// TIA Portal V17 export
// export: Created 2026-04-13T11:12:44.8952859Z, ExportSetting WithDefaults, DisplayName Totally Integrated Automation Portal, DisplayVersion V17 Update 4, DisplayName TIA Portal Openness, DisplayVersion V17 Update 4, DisplayName TIA Portal Version Control Interface, DisplayVersion V17, DisplayName SINAMICS Startdrive Advanced, DisplayVersion V17, DisplayName SINAMICS Startdrive G130, G150, S120, S150, SINAMICS MV, S210, DisplayVersion V17, DisplayName SINAMICS Startdrive G110M, G120, G120C, G120D, G120P, G115D, DisplayVersion V17, DisplayName STEP 7 Professional, DisplayVersion V17 Update 4, DisplayName STEP 7 Safety, DisplayVersion V17, DisplayName WinCC Professional, DisplayVersion V17 Update 4
FUNCTION_BLOCK "Send_Config"   // FB611, SCL
TITLE = Send Configuration
AUTHOR : SIMATIC
FAMILY : Freeport
NAME : SendConf
VERSION : 4.0
// stored: IsIECCheckEnabled false, SetENOAutomatically false, UDAEnableTagReadback false
   VAR_INPUT
      REQ : Bool;   // Startet die Konfiguration für Senden bei steigender Flanke / Activates the configuration for sending on rising edge
      PORT : PORT := 0;   // Kommunikationsport, Hardwarekennung / Communication port, Hardware Identifier
      RTSONDLY : UInt := 16#00;   // Wartezeit nach Aktivierung von RTS, vor Übertragung von Tx-Daten (ms) / Time to wait after activating RTS before transmission will be initiated (ms)
      RTSOFFDLY : UInt := 16#00;   // Wartezeit nach Übertragung von Tx-Daten, bevor RTS deaktiviert wird (ms) / Time to wait before de-activating RTS once transmission has been completed (ms)
      BREAK : UInt := 16#00;   // Pause vor Start jeder Übertragung (Bitzeiten) / On start of a message, a break will be sent for the specified no. of bit times
      IDLELINE : UInt := 16#00;   // Leerlaufzeit vor Start jeder Übertragung (Bitzeiten) / Number of bits times the line will be idle before the next transmission
      USR_END : String[2] := '';   // Anzahl der Endekennzeichen / Number of characters in the end delimiter
      APP_END : String[5] := '';   // Anzahl angehängter Zeichen / Number of characters to be appended to the transmitted message
   END_VAR
   VAR_OUTPUT
      DONE : Bool;   // Anweisung beendet ohne Fehler / Instruction finished without error
      ERROR : Bool;   // Anweisung beendet mit Fehler / Instruction finished with error
      STATUS : Word := W#16#7000;   // Zusätzliche Fehlerinformation / Detailed error information
   END_VAR
   VAR
      b_e_REQ : Bool;   // Flankenbit für REQ / Edge flag for REQ
      y_state : SInt := 16#00;   // Status der Anweisung / State of instruction
      WRREC { S7_SetPoint := 'True'} : WRREC;   // Lokale Instanz der Anweisung WRREC / Local instance of instruction WRREC
      RDREC { S7_SetPoint := 'True'} : RDREC;   // Lokale Instanz der Anweisung RDREC / Local instance of instruction RDREC
      w_record { S7_SetPoint := 'True'} : P2P_SendCfgData;   // Nur für internen Gebrauch / For internal use only
      r_record { S7_SetPoint := 'True'} : P2P_RdEstat;   // Nur für internen Gebrauch / For internal use only
   END_VAR
BEGIN
END_FUNCTION_BLOCK
